// TIA Portal project "Styringsenhed" (V13)

(* hardware
DEVICE "S7-1200 station_1"  S7-1200 Station
   slot 0: "Rack_0"  Rack  V1.0
   slot 1: "PLC_1"  CPU 1214C DC/DC/DC  6ES7 214-1AG40-0XB0  V4.1
   slot 3: "AQ 1x12BIT_1"  6ES7 232-4HA30-0XB0  V1.0
DEVICE "HMI_1"  KTP700 Basic PN
   slot 0: "HMI"  HMI  6AV2 123-2GB03-0AX0  13.0.1.0
   slot 1: "HMI_RT_1"  KTP700 Basic PN  6AV2 123-2GB03-0AX0  13.0.1.0
   slot 5: "HMI_1.IE_CP_1"  PROFINET Interface
      slot 1: "PROFINET Interface_1"  PROFINET Interface
         slot 1: "Port_1"  Port
*)

// ===== PLC "PLC_1"  CPU 1214C DC/DC/DC =====

VAR_GLOBAL   // PLC tag table "Default tag table"
   "Trin1" AT %Q0.6 : Bool;
   "Trin2" AT %Q0.7 : Bool;
   "Trin3" AT %Q1.0 : Bool;
   "SpændingCentral" AT %MB0 : USInt;
   "ManuelMode" AT %I0.0 : Bool;
   "KnapOp" AT %I0.1 : Bool;
   "KnapNed" AT %I0.2 : Bool;
END_VAR

DATA_BLOCK "Trinskifter_DB"   // DB8
{ S7_Optimized_Access := 'FALSE' }
VERSION : 0.1
// stored: InstanceOfName Trinskifter
"Trinskifter"
BEGIN
END_DATA_BLOCK

DATA_BLOCK "Ethernet"   // DB14
{ S7_Optimized_Access := 'FALSE' }
VERSION : 0.1
   VAR
      EnableForbindelse : Bool;
      EnableSend : Bool;
      EnableModtag : Bool;
      DisableForbindelse : Bool;
      SendData : Array[0..3] of Char;
      ModtagData : Array[0..3] of Word;
      EnhedToReq : USInt;
      Req1 : Array[0..3] of Char;
      Req2 : Array[0..3] of Char;
      Firsttime : Bool;
      Invert : Bool;
   END_VAR
BEGIN
END_DATA_BLOCK

DATA_BLOCK "HMI"   // DB21
{ S7_Optimized_Access := 'FALSE' }
VERSION : 0.1
   VAR
      DataCentralEnhed : Array[0..3] of Word;
      DataDecentralEnhed : Array[0..3] of Word;
   END_VAR
BEGIN
END_DATA_BLOCK

// folder: System blocks/Program resources

DATA_BLOCK "ManTrinskift1til2"   // DB1
{ S7_Optimized_Access := 'FALSE' }
AUTHOR : Simatic
FAMILY : IEC
NAME : IEC_TMR
VERSION : 1.0
// stored: InstanceOfName ?
"?"
BEGIN
END_DATA_BLOCK

DATA_BLOCK "Trinskift2til1"   // DB2
{ S7_Optimized_Access := 'FALSE' }
AUTHOR : Simatic
FAMILY : IEC
NAME : IEC_TMR
VERSION : 1.0
// stored: InstanceOfName ?
"?"
BEGIN
END_DATA_BLOCK

DATA_BLOCK "Trinskift2til3"   // DB3
{ S7_Optimized_Access := 'FALSE' }
AUTHOR : Simatic
FAMILY : IEC
NAME : IEC_TMR
VERSION : 1.0
// stored: InstanceOfName ?
"?"
BEGIN
END_DATA_BLOCK

DATA_BLOCK "Trinskift1til2"   // DB4
{ S7_Optimized_Access := 'FALSE' }
AUTHOR : Simatic
FAMILY : IEC
NAME : IEC_TMR
VERSION : 1.0
// stored: InstanceOfName ?
"?"
BEGIN
END_DATA_BLOCK

DATA_BLOCK "Trinskift3til2"   // DB5
{ S7_Optimized_Access := 'FALSE' }
AUTHOR : Simatic
FAMILY : IEC
NAME : IEC_TMR
VERSION : 1.0
// stored: InstanceOfName ?
"?"
BEGIN
END_DATA_BLOCK

DATA_BLOCK "Trin1VentTilNyData"   // DB6
{ S7_Optimized_Access := 'FALSE' }
AUTHOR : Simatic
FAMILY : IEC
NAME : IEC_TMR
VERSION : 1.0
// stored: InstanceOfName ?
"?"
BEGIN
END_DATA_BLOCK

DATA_BLOCK "Trin2VentTilNyData"   // DB7
{ S7_Optimized_Access := 'FALSE' }
AUTHOR : Simatic
FAMILY : IEC
NAME : IEC_TMR
VERSION : 1.0
// stored: InstanceOfName ?
"?"
BEGIN
END_DATA_BLOCK

DATA_BLOCK "ManTrinskift2til3"   // DB9
{ S7_Optimized_Access := 'FALSE' }
AUTHOR : Simatic
FAMILY : IEC
NAME : IEC_TMR
VERSION : 1.0
// stored: InstanceOfName ?
"?"
BEGIN
END_DATA_BLOCK

DATA_BLOCK "ManTrinskift2til1"   // DB10
{ S7_Optimized_Access := 'FALSE' }
AUTHOR : Simatic
FAMILY : IEC
NAME : IEC_TMR
VERSION : 1.0
// stored: InstanceOfName ?
"?"
BEGIN
END_DATA_BLOCK

DATA_BLOCK "Trin3VentTilNyData"   // DB11
{ S7_Optimized_Access := 'FALSE' }
AUTHOR : Simatic
FAMILY : IEC
NAME : IEC_TMR
VERSION : 1.0
// stored: InstanceOfName ?
"?"
BEGIN
END_DATA_BLOCK

DATA_BLOCK "ManTrinskift3til2"   // DB12
{ S7_Optimized_Access := 'FALSE' }
AUTHOR : Simatic
FAMILY : IEC
NAME : IEC_TMR
VERSION : 1.0
// stored: InstanceOfName ?
"?"
BEGIN
END_DATA_BLOCK

DATA_BLOCK "PLC_1_Connection_DB"   // DB16
{ S7_Optimized_Access := 'FALSE' }
AUTHOR : SIMATIC
FAMILY : MC7Plus
NAME : TC_IP_v4
VERSION : 1.0
// stored: InstanceOfName ?
"?"
BEGIN
END_DATA_BLOCK

DATA_BLOCK "SendDataTimer"   // DB20
{ S7_Optimized_Access := 'FALSE' }
AUTHOR : Simatic
FAMILY : IEC
NAME : IEC_TMR
VERSION : 1.0
// stored: InstanceOfName ?
"?"
BEGIN
END_DATA_BLOCK

DATA_BLOCK "ModtagDataTimer"   // DB22
{ S7_Optimized_Access := 'FALSE' }
AUTHOR : Simatic
FAMILY : IEC
NAME : IEC_TMR
VERSION : 1.0
// stored: InstanceOfName ?
"?"
BEGIN
END_DATA_BLOCK

// folder: (top level)

FUNCTION_BLOCK "Trinskifter"   // FB1, LAD
{ S7_Optimized_Access := 'FALSE' }
VERSION : 0.1
   VAR_TEMP   // added for the SCL form of the ladder/FBD networks
      _w1 : Bool;
      _w2 : Bool;
   END_VAR
BEGIN

REGION Network 1: Start
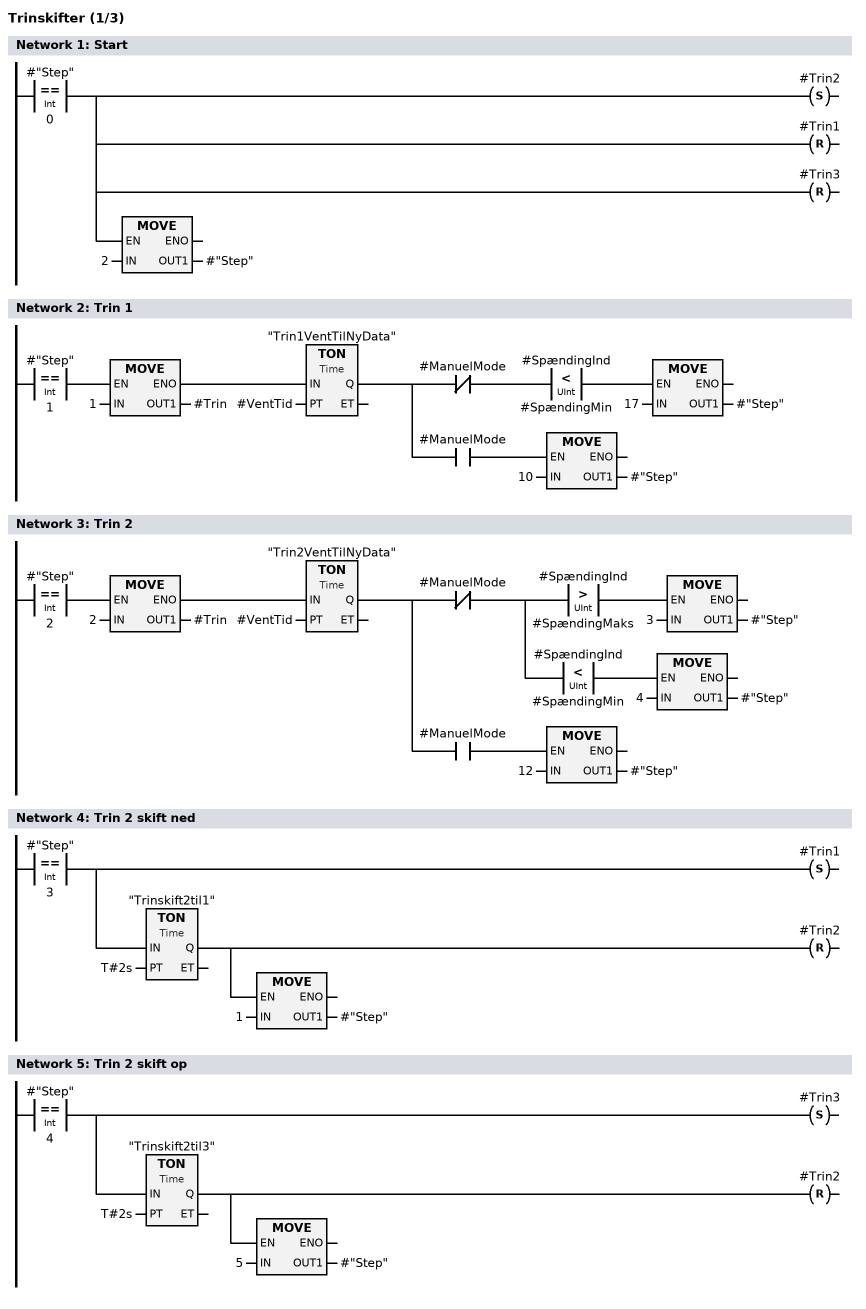
   RUNG wire#powerrail
      { S7_Templates := "SrcType := Int" } EQ_Contact(in1 := #"Step", in2 := 0)
      wire#w1
      S_Coil( #Trin2 )
   END_RUNG
   RUNG wire#w1
      R_Coil( #Trin1 )
   END_RUNG
   RUNG wire#w1
      R_Coil( #Trin3 )
   END_RUNG
   RUNG wire#w1
      Move(in := 2, out1 => #"Step")
   END_RUNG
   // the same network as SCL:
   IF #"Step" = 0 THEN
       #Trin2 := TRUE;
       #Trin1 := FALSE;
       #Trin3 := FALSE;
       #"Step" := 2;
   END_IF;
END_REGION

REGION Network 2: Trin 1
   #_w1 := #"Step" = 1;
   IF #_w1 THEN #Trin := 1; END_IF;
   "Trin1VentTilNyData".TON(IN := #_w1, PT := #VentTid);
   IF "Trin1VentTilNyData".Q AND NOT #ManuelMode AND (#SpændingInd < #SpændingMin) THEN
       #"Step" := 17;
   END_IF;
   IF "Trin1VentTilNyData".Q AND #ManuelMode THEN #"Step" := 10; END_IF;
END_REGION

REGION Network 3: Trin 2
   #_w1 := #"Step" = 2;
   IF #_w1 THEN #Trin := 2; END_IF;
   "Trin2VentTilNyData".TON(IN := #_w1, PT := #VentTid);
   #_w2 := "Trin2VentTilNyData".Q AND NOT #ManuelMode;
   IF #_w2 AND (#SpændingInd > #SpændingMaks) THEN #"Step" := 3; END_IF;
   IF #_w2 AND (#SpændingInd < #SpændingMin) THEN #"Step" := 4; END_IF;
   IF "Trin2VentTilNyData".Q AND #ManuelMode THEN #"Step" := 12; END_IF;
END_REGION

REGION Network 4: Trin 2 skift ned
   #_w1 := #"Step" = 3;
   IF #_w1 THEN #Trin1 := TRUE; END_IF;
   "Trinskift2til1".TON(IN := #_w1, PT := T#2s);
   IF "Trinskift2til1".Q THEN
       #Trin2 := FALSE;
       #"Step" := 1;
   END_IF;
END_REGION

REGION Network 5: Trin 2 skift op
   #_w1 := #"Step" = 4;
   IF #_w1 THEN #Trin3 := TRUE; END_IF;
   "Trinskift2til3".TON(IN := #_w1, PT := T#2s);
   IF "Trinskift2til3".Q THEN
       #Trin2 := FALSE;
       #"Step" := 5;
   END_IF;
END_REGION

REGION Network 6: Trin 3
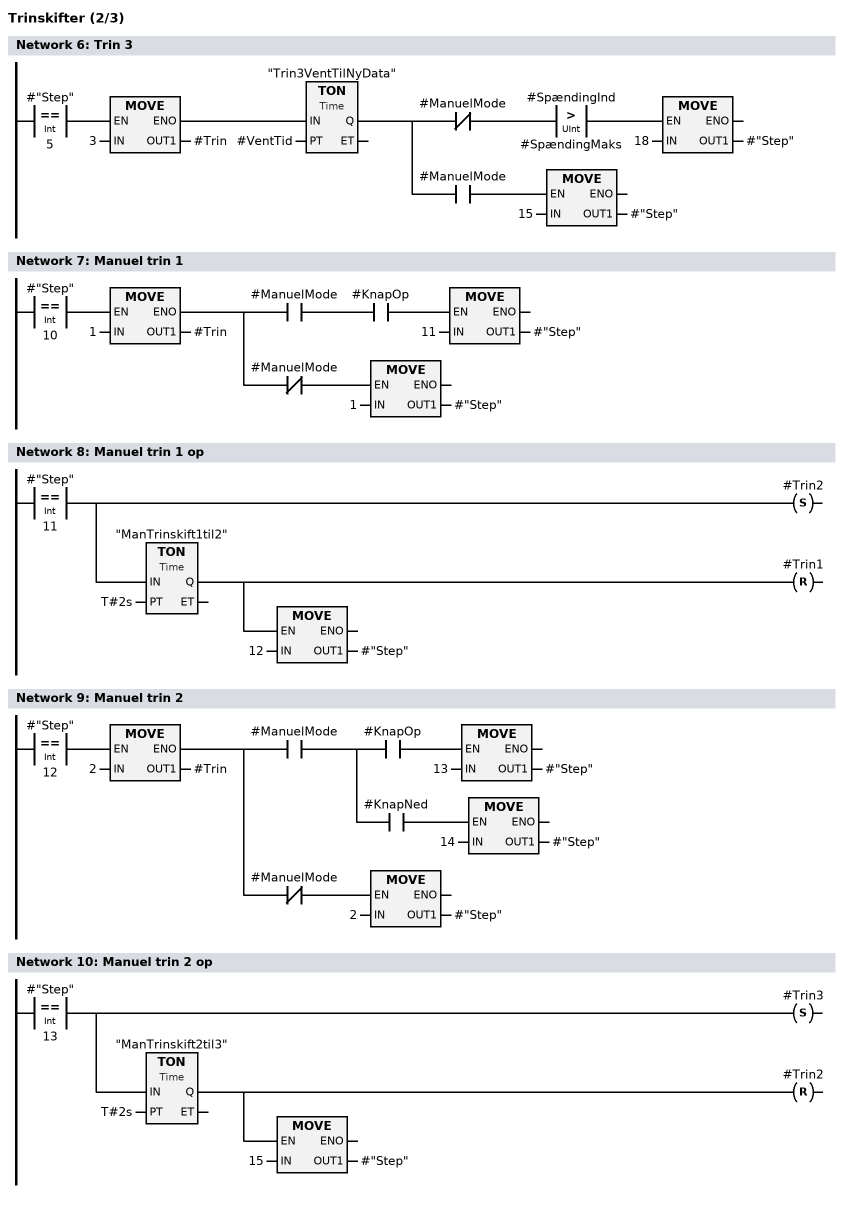
   #_w1 := #"Step" = 5;
   IF #_w1 THEN #Trin := 3; END_IF;
   "Trin3VentTilNyData".TON(IN := #_w1, PT := #VentTid);
   IF "Trin3VentTilNyData".Q AND NOT #ManuelMode AND (#SpændingInd > #SpændingMaks) THEN
       #"Step" := 18;
   END_IF;
   IF "Trin3VentTilNyData".Q AND #ManuelMode THEN #"Step" := 15; END_IF;
END_REGION

REGION Network 7: Manuel trin 1
   RUNG wire#powerrail
      { S7_Templates := "SrcType := Int" } EQ_Contact(in1 := #"Step", in2 := 10)
      Move(in := 1, out1 => #Trin)
      wire#w1
      Contact( #ManuelMode )
      Contact( #KnapOp )
      Move(in := 11, out1 => #"Step")
   END_RUNG
   RUNG wire#w1
      I_Contact( #ManuelMode )
      Move(in := 1, out1 => #"Step")
   END_RUNG
   // the same network as SCL:
   #_w1 := #"Step" = 10;
   IF #_w1 THEN #Trin := 1; END_IF;
   IF #_w1 AND #ManuelMode AND #KnapOp THEN #"Step" := 11; END_IF;
   IF #_w1 AND NOT #ManuelMode THEN #"Step" := 1; END_IF;
END_REGION

REGION Network 8: Manuel trin 1 op
   #_w1 := #"Step" = 11;
   IF #_w1 THEN #Trin2 := TRUE; END_IF;
   "ManTrinskift1til2".TON(IN := #_w1, PT := T#2s);
   IF "ManTrinskift1til2".Q THEN
       #Trin1 := FALSE;
       #"Step" := 12;
   END_IF;
END_REGION

REGION Network 9: Manuel trin 2
   RUNG wire#powerrail
      { S7_Templates := "SrcType := Int" } EQ_Contact(in1 := #"Step", in2 := 12)
      Move(in := 2, out1 => #Trin)
      wire#w1
      Contact( #ManuelMode )
      wire#w2
      Contact( #KnapOp )
      Move(in := 13, out1 => #"Step")
   END_RUNG
   RUNG wire#w2
      Contact( #KnapNed )
      Move(in := 14, out1 => #"Step")
   END_RUNG
   RUNG wire#w1
      I_Contact( #ManuelMode )
      Move(in := 2, out1 => #"Step")
   END_RUNG
   // the same network as SCL:
   #_w1 := #"Step" = 12;
   IF #_w1 THEN #Trin := 2; END_IF;
   #_w2 := #_w1 AND #ManuelMode;
   IF #_w2 AND #KnapOp THEN #"Step" := 13; END_IF;
   IF #_w2 AND #KnapNed THEN #"Step" := 14; END_IF;
   IF #_w1 AND NOT #ManuelMode THEN #"Step" := 2; END_IF;
END_REGION

REGION Network 10: Manuel trin 2 op
   #_w1 := #"Step" = 13;
   IF #_w1 THEN #Trin3 := TRUE; END_IF;
   "ManTrinskift2til3".TON(IN := #_w1, PT := T#2s);
   IF "ManTrinskift2til3".Q THEN
       #Trin2 := FALSE;
       #"Step" := 15;
   END_IF;
END_REGION

REGION Network 11: Manuel trin 2 ned
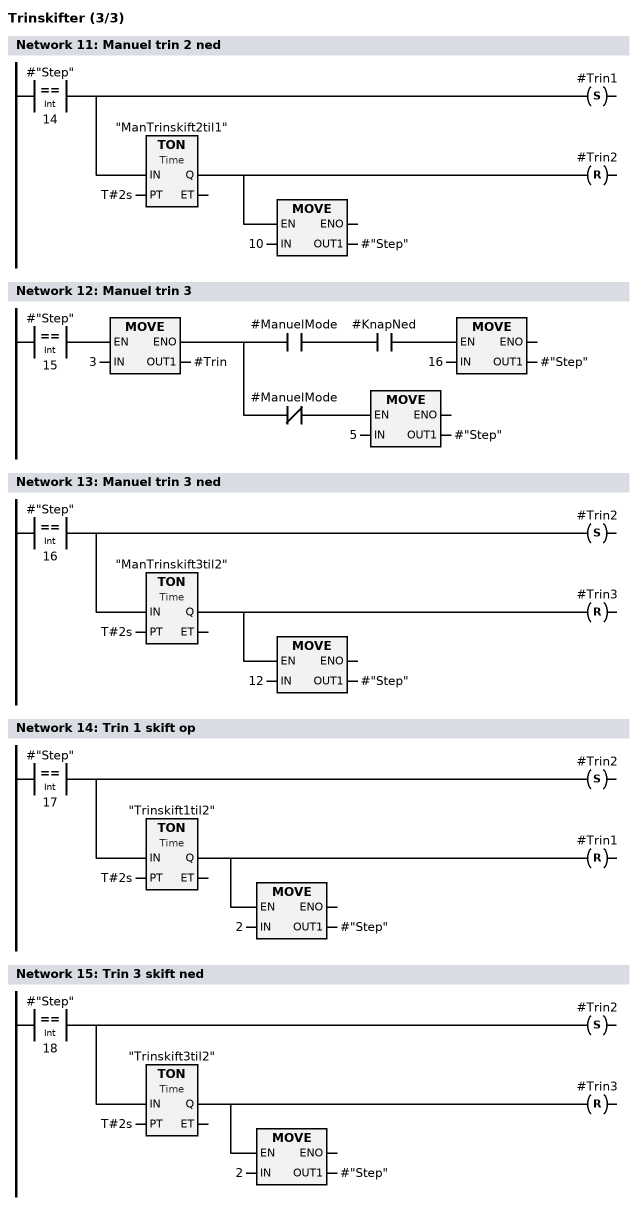
   #_w1 := #"Step" = 14;
   IF #_w1 THEN #Trin1 := TRUE; END_IF;
   "ManTrinskift2til1".TON(IN := #_w1, PT := T#2s);
   IF "ManTrinskift2til1".Q THEN
       #Trin2 := FALSE;
       #"Step" := 10;
   END_IF;
END_REGION

REGION Network 12: Manuel trin 3
   RUNG wire#powerrail
      { S7_Templates := "SrcType := Int" } EQ_Contact(in1 := #"Step", in2 := 15)
      Move(in := 3, out1 => #Trin)
      wire#w1
      Contact( #ManuelMode )
      Contact( #KnapNed )
      Move(in := 16, out1 => #"Step")
   END_RUNG
   RUNG wire#w1
      I_Contact( #ManuelMode )
      Move(in := 5, out1 => #"Step")
   END_RUNG
   // the same network as SCL:
   #_w1 := #"Step" = 15;
   IF #_w1 THEN #Trin := 3; END_IF;
   IF #_w1 AND #ManuelMode AND #KnapNed THEN #"Step" := 16; END_IF;
   IF #_w1 AND NOT #ManuelMode THEN #"Step" := 5; END_IF;
END_REGION

REGION Network 13: Manuel trin 3 ned
   #_w1 := #"Step" = 16;
   IF #_w1 THEN #Trin2 := TRUE; END_IF;
   "ManTrinskift3til2".TON(IN := #_w1, PT := T#2s);
   IF "ManTrinskift3til2".Q THEN
       #Trin3 := FALSE;
       #"Step" := 12;
   END_IF;
END_REGION

REGION Network 14: Trin 1 skift op
   #_w1 := #"Step" = 17;
   IF #_w1 THEN #Trin2 := TRUE; END_IF;
   "Trinskift1til2".TON(IN := #_w1, PT := T#2s);
   IF "Trinskift1til2".Q THEN
       #Trin1 := FALSE;
       #"Step" := 2;
   END_IF;
END_REGION

REGION Network 15: Trin 3 skift ned
   #_w1 := #"Step" = 18;
   IF #_w1 THEN #Trin2 := TRUE; END_IF;
   "Trinskift3til2".TON(IN := #_w1, PT := T#2s);
   IF "Trinskift3til2".Q THEN
       #Trin3 := FALSE;
       #"Step" := 2;
   END_IF;
END_REGION
END_FUNCTION_BLOCK

FUNCTION "OpretForbindelse" : Void   // FC1, LAD
{ S7_Optimized_Access := 'FALSE' }
VERSION : 0.1
BEGIN

REGION Network 1: TCON
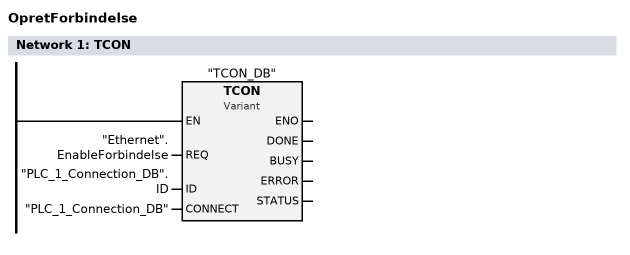
   "TCON_DB"(REQ := "Ethernet".EnableForbindelse,   // TCON
             ID := "PLC_1_Connection_DB".ID,
             CONNECT := "PLC_1_Connection_DB");
END_REGION
END_FUNCTION

FUNCTION "SendData" : Void   // FC2, LAD
{ S7_Optimized_Access := 'FALSE' }
VERSION : 0.1
BEGIN

REGION Network 1: Vælg enhed til data request
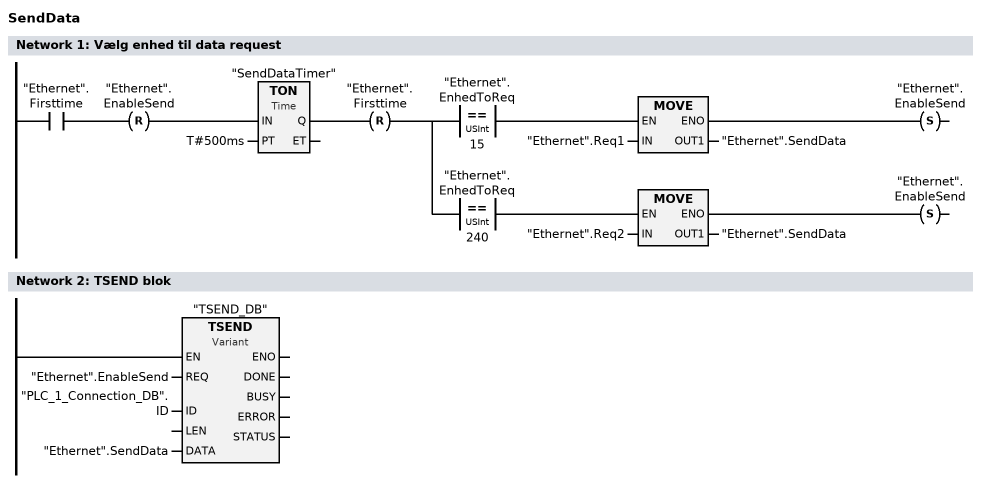
   IF "Ethernet".Firsttime THEN "Ethernet".EnableSend := FALSE; END_IF;
   "SendDataTimer".TON(IN := "Ethernet".Firsttime, PT := T#500ms);
   IF "SendDataTimer".Q THEN "Ethernet".Firsttime := FALSE; END_IF;
   IF "SendDataTimer".Q AND ("Ethernet".EnhedToReq = 15) THEN
       "Ethernet".SendData := "Ethernet".Req1;
       "Ethernet".EnableSend := TRUE;
   END_IF;
   IF "SendDataTimer".Q AND ("Ethernet".EnhedToReq = 240) THEN
       "Ethernet".SendData := "Ethernet".Req2;
       "Ethernet".EnableSend := TRUE;
   END_IF;
END_REGION

REGION Network 2: TSEND blok
   "TSEND_DB"(REQ := "Ethernet".EnableSend, ID := "PLC_1_Connection_DB".ID, DATA := "Ethernet".SendData);   // TSEND
END_REGION
END_FUNCTION

FUNCTION "ModtagData" : Void   // FC3, LAD
{ S7_Optimized_Access := 'FALSE' }
VERSION : 0.1
BEGIN

REGION Network 1: TRCV
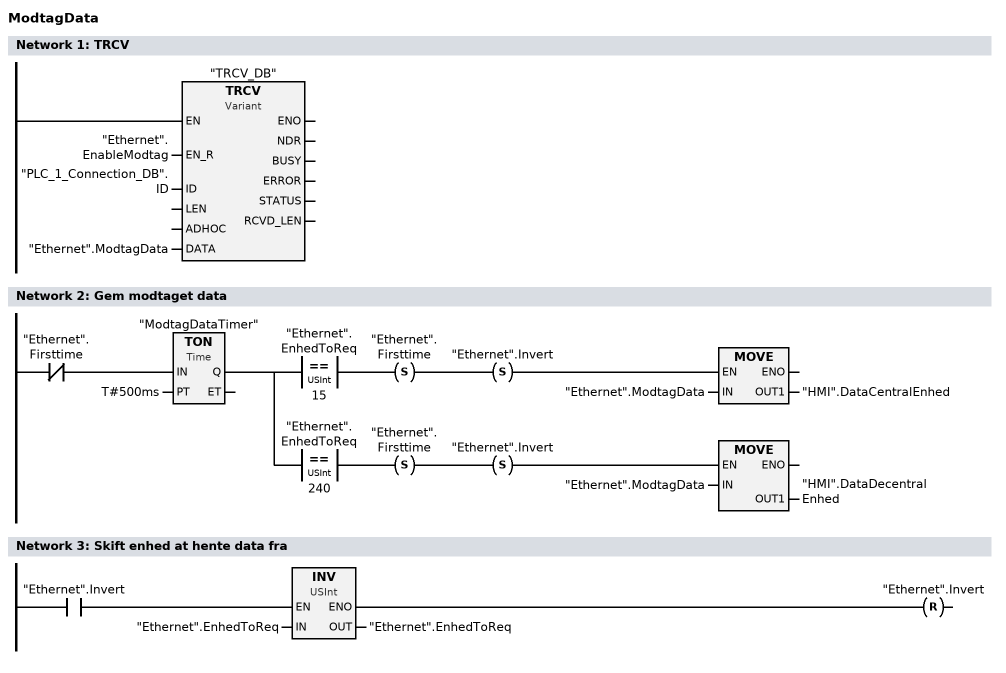
   "TRCV_DB"(EN_R := "Ethernet".EnableModtag, ID := "PLC_1_Connection_DB".ID, DATA := "Ethernet".ModtagData);   // TRCV
END_REGION

REGION Network 2: Gem modtaget data
   "ModtagDataTimer".TON(IN := NOT "Ethernet".Firsttime, PT := T#500ms);
   IF "ModtagDataTimer".Q AND ("Ethernet".EnhedToReq = 15) THEN
       "Ethernet".Firsttime := TRUE;
       "Ethernet".Invert := TRUE;
       "HMI".DataCentralEnhed := "Ethernet".ModtagData;
   END_IF;
   IF "ModtagDataTimer".Q AND ("Ethernet".EnhedToReq = 240) THEN
       "Ethernet".Firsttime := TRUE;
       "Ethernet".Invert := TRUE;
       "HMI".DataDecentralEnhed := "Ethernet".ModtagData;
   END_IF;
END_REGION

REGION Network 3: Skift enhed at hente data fra
   RUNG wire#powerrail
      Contact( "Ethernet".Invert )
      { S7_Templates := "SrcType := USInt" } Inv(in := "Ethernet".EnhedToReq, out => "Ethernet".EnhedToReq)
      R_Coil( "Ethernet".Invert )
   END_RUNG
   // the same network as SCL:
   IF "Ethernet".Invert THEN
       "Ethernet".EnhedToReq := NOT "Ethernet".EnhedToReq;
       "Ethernet".Invert := FALSE;
   END_IF;
END_REGION
END_FUNCTION

FUNCTION "AfslutForbindelse" : Void   // FC4, LAD
{ S7_Optimized_Access := 'FALSE' }
VERSION : 0.1
BEGIN

REGION Network 1: TDISCON
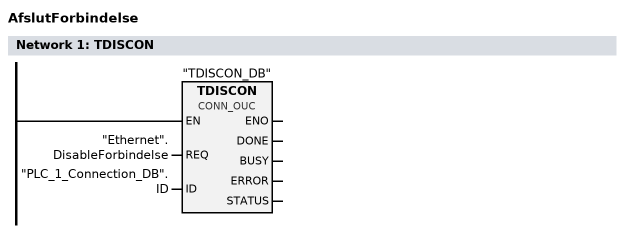
   "TDISCON_DB"(REQ := "Ethernet".DisableForbindelse, ID := "PLC_1_Connection_DB".ID);   // TDISCON
END_REGION
END_FUNCTION

ORGANIZATION_BLOCK "Main"   // OB1, LAD, ProgramCycle
TITLE = "Main Program Sweep (Cycle)"
{ S7_Optimized_Access := 'FALSE' }
VERSION : 0.1
BEGIN

REGION Network 1: Trinskift
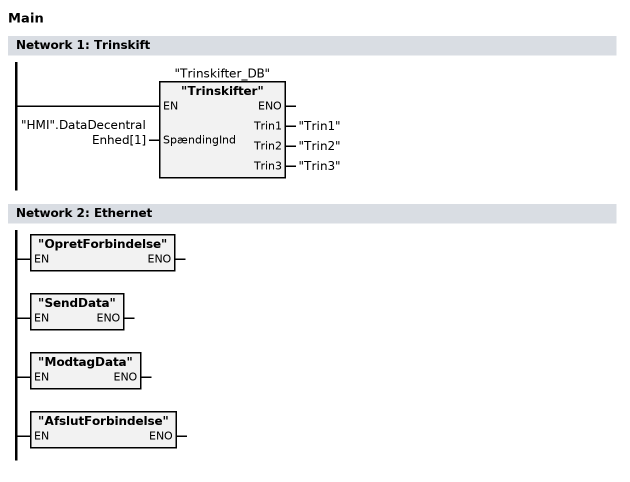
   RUNG wire#powerrail
      "Trinskifter_DB"(SpændingInd := "HMI".DataDecentralEnhed[1], Trin1 => "Trin1", Trin2 => "Trin2", Trin3 => "Trin3")
   END_RUNG
   // the same network as SCL:
   "Trinskifter_DB"(SpændingInd := "HMI".DataDecentralEnhed[1],   // "Trinskifter"
                    Trin1 => "Trin1",
                    Trin2 => "Trin2",
                    Trin3 => "Trin3");
END_REGION

REGION Network 2: Ethernet
   RUNG wire#powerrail
      "OpretForbindelse"()
   END_RUNG
   RUNG wire#powerrail
      "SendData"()
   END_RUNG
   RUNG wire#powerrail
      "ModtagData"()
   END_RUNG
   RUNG wire#powerrail
      "AfslutForbindelse"()
   END_RUNG
   // the same network as SCL:
   "OpretForbindelse"();
   "SendData"();
   "ModtagData"();
   "AfslutForbindelse"();
END_REGION
END_ORGANIZATION_BLOCK

(* ===== HMI "HMI_RT_1" =====
connection "HMI_Connection_1": ETHERNET, SMART_S7_1200_OMS

HMI tags "Default tag table"
   "Tag_ScreenNumber" : UInt, internal
   "HMI_KnapOp" : Bool, 1 s
   "HMI_KnapNed" : Bool, 1 s
   "HMI_Trin" : Int, 1 s
   "HMI_StrømCentral" : Word, 1 s
   "HMI_ManuelMode" : Bool, 1 s
   "HMI_SpændingCentral" : Word, 1 s
   "HMI_THDCentral" : Word, 1 s
   "HMI_StrømForbruger1" : Word, 1 s
   "HMI_SpændingForbruger1" : Word, 1 s
   "HMI_THDForbruger1" : Word, 1 s
   "HMI_PowerfactorCentral" : Word, 1 s
   "HMI_PowerfactorForbruger1" : Word, 1 s

Template "Template_1" 800x480
   Button "Template_Button" at 266,202 size 52x37
   Button "Template_Button_1" at 213,202 size 52x37
   Button "Template_Button_2" at 160,202 size 52x37
   Button "Template_Button_3" at 107,202 size 52x37
   Button "Template_Button_4" at 54,202 size 52x37
   Button "Template_Button_5" at 1,202 size 52x37
   SymbolicIOField "Symbolic_IO_Field_Screen" at 69,7 size 164x24
   DateTimeField "HmiScreenItemData" at 235,19 size 85x19
   DateTimeField "HmiScreenItemData_1" at 235,0 size 85x19
   GraphicView "Logo" at 0,0 size 67x38

screen "Root screen" 800x480, template "Template_1"
   TextField "HmiScreenItemData" at 32,112 size 256x17

screen "Automatisk mode" 800x480
   TextField "Text field_1" at 211,20 size 428x60
   TextField "Text field_12" at 264,453 size 262x27
   TextField "Text field_9" at 495,361 size 170x43
   IOField "I/O field_10" at 495,404 size 170x38
   Button "Button_1" at 186,387 size 104x54
   Button "Button_2" at 50,387 size 104x54
   TextField "Text field_2" at 416,74 size 144x67
   TextField "Text field_3" at 600,74 size 144x67
   TextField "Text field_4" at 209,79 size 167x66
   TextField "Text field_5" at 50,257 size 132x27
   TextField "Text field_6" at 50,157 size 66x27
   TextField "Text field_7" at 50,207 size 106x27
   IOField "I/O field_4" at 606,149 size 116x38
   IOField "I/O field_5" at 606,202 size 116x38
   IOField "I/O field_6" at 606,255 size 116x38
   TextField "Text field_8" at 50,308 size 47x27
   IOField "I/O field_11" at 606,308 size 116x38
   IOField "I/O field_7" at 413,152 size 116x38
   IOField "I/O field_1" at 413,204 size 116x38
   IOField "I/O field_2" at 413,256 size 116x38
   IOField "I/O field_3" at 206,152 size 116x38
   IOField "I/O field_8" at 206,204 size 116x38
   IOField "I/O field_9" at 206,256 size 116x38
   IOField "I/O field_12" at 413,308 size 116x38
   IOField "I/O field_13" at 206,308 size 116x38

screen "Manuel mode" 800x480
   TextField "Text field_9" at 495,361 size 170x43
   IOField "I/O field_10" at 495,404 size 170x38
   Button "Button_1" at 186,387 size 104x54
   Button "Button_2" at 50,387 size 104x54
   TextField "Text field_12" at 264,453 size 307x27
   TextField "Text field_1" at 255,20 size 328x60
   TextField "Text field_2" at 416,74 size 144x67
   TextField "Text field_4" at 209,79 size 167x66
   TextField "Text field_5" at 50,257 size 132x27
   TextField "Text field_6" at 50,157 size 66x27
   TextField "Text field_7" at 50,207 size 106x27
   IOField "I/O field_4" at 606,149 size 116x38
   IOField "I/O field_5" at 606,202 size 116x38
   IOField "I/O field_6" at 606,255 size 116x38
   TextField "Text field_8" at 50,308 size 47x27
   IOField "I/O field_11" at 606,308 size 116x38
   IOField "I/O field_7" at 413,152 size 116x38
   IOField "I/O field_1" at 413,204 size 116x38
   IOField "I/O field_2" at 413,256 size 116x38
   IOField "I/O field_3" at 206,152 size 116x38
   IOField "I/O field_8" at 206,204 size 116x38
   IOField "I/O field_9" at 206,256 size 116x38
   IOField "I/O field_12" at 413,308 size 116x38
   IOField "I/O field_13" at 206,308 size 116x38
   TextField "Text field_3" at 600,74 size 144x67
*)